(* CoDeSys 2.3.9.41 project: hlor.pro *)
(* Libraries: STANDARD.LIB 4.10.05 11:14:46, IECSFC.LIB 13.4.06 15:51:28, ANALYZATION.LIB 5.10.99 09:05:06 *)

(* PLC configuration (modules and I/O channels)
AT %IX0.0 [BitInput] {ChannellName = Enter name}
AT %IX0.1 [BitInput] {ChannellName = Enter name}
AT %IX0.2 [BitInput] {ChannellName = Enter name}
AT %IX0.3 [BitInput] {ChannellName = Enter name}
AT %IB1.0 [ByteInput] {ChannellName = Enter name}
AT %IB1.1 [ByteInput] {ChannellName = Enter name}
SolNasos AT %QX2.0 [BitOutput] Вкл/Выкл солевого насоса {ChannellName = Enter name}
WaterNasos AT %QX2.1 [BitOutput] Вкл/Выкл насоса воды {ChannellName = Enter name}
Klapan AT %QX2.2 [BitOutput] Вкл/Выкл клапана воды {ChannellName = Enter name}
Elektroliz AT %QX2.3 [BitOutput] Вкл/Выкл выпрямителя {ChannellName = Enter name}
AT %QB3.0 [ByteOutput] {ChannellName = Enter name}
AT %QB3.1 [ByteOutput] {ChannellName = Enter name}
D_Volume_Bak AT %IR4.0 [FloatInputP] Объем бака {ChannellName = Fast analog input; AIN_TYPE = 4-20 mA; Peak_Filtr = 200; Flt_Ch = Off; TauRC = 10; MinFV = 0; MaxFV = 150}
D_Konduktivnost AT %IR4.1 [FloatInputP] D_Konduktivnost {ChannellName = Fast analog input; AIN_TYPE = 4-20 mA; Peak_Filtr = 200; Flt_Ch = Off; TauRC = 10; MinFV = 0; MaxFV = 200}
D_Volt AT %IR4.2 [FloatInputP] Ток выпрямителя {ChannellName = Fast analog input; AIN_TYPE = 4-20 mA; Peak_Filtr = 200; Flt_Ch = Off; TauRC = 10; MinFV = 0; MaxFV = 80}
D_Amper AT %IR4.3 [FloatInputP] Напряжение выпрямителя {ChannellName = Fast analog input; AIN_TYPE = 4-20 mA; Peak_Filtr = 200; Flt_Ch = Off; TauRC = 10; MinFV = 0; MaxFV = 200}
DT_Water_Input AT %IR4.4 [FloatInputP] Температура воды на входе {ChannellName = Fast analog input; AIN_TYPE = 4-20 mA; Peak_Filtr = 200; Flt_Ch = Off; TauRC = 10; MinFV = 0; MaxFV = 100}
DT_Water_output AT %IR4.5 [FloatInputP] Температура воды на выходе {ChannellName = Fast analog input; AIN_TYPE = 4-20 mA; Peak_Filtr = 200; Flt_Ch = Off; TauRC = 10; MinFV = 0; MaxFV = 100}
AT %IR4.6 [FloatInputP] {ChannellName = Fast analog input; AIN_TYPE = 4-20 mA; Peak_Filtr = 200; Flt_Ch = Off; TauRC = 10; MinFV = 0; MaxFV = 100}
AT %IR4.7 [FloatInputP] {ChannellName = Fast analog input; AIN_TYPE = 4-20 mA; Peak_Filtr = 200; Flt_Ch = Off; TauRC = 10; MinFV = 0; MaxFV = 20000.0}
AT %IW4.8 [WordInput] {ChannellName = Enter name}
AT %QR5.0 [FloatOutputP] {ChannellName = Analog output; AOUT_TYPE = 4-20 mA; SafeValueREAL = 0.0}
AT %QR5.1 [FloatOutputP] {ChannellName = Analog output; AOUT_TYPE = 4-20 mA; SafeValueREAL = 0.0}
AT %QR5.2 [FloatOutputP] {ChannellName = Analog output; AOUT_TYPE = 4-20 mA; SafeValueREAL = 0.0}
AT %QR5.3 [FloatOutputP] {ChannellName = Analog output; AOUT_TYPE = 4-20 mA; SafeValueREAL = 0.0}
Special input [ID103] node 6, in %IB6 out %QB6 {ChannellName = Special input}
  AT %IX6.0 [BitInput] {ChannellName = Enter name}
Special output [ID104] node 7, in %IB7 out %QB7 {ChannellName = Special output}
  AT %QX7.0 [BitOutput] {ChannellName = Enter name}
Modbus [MODBUS_ID302] node 0, in %IB8.0 out %QB8.0 {ChannellName = Modbus}
  TCP [TCP_ID221] node 0, in %IB8.0.0 out %QB8.0.0 {ChannellName = TCP; RemotePort = 502; Visibility = No}
8 bits [8Bit] node 1, in %IB8.1 out %QB8.1 {ChannellName = 8 bit}
  AT %QB8.1.0 [ByteOutput] {ChannellName = Enter name}
8 bits [8Bit] node 2, in %IB8.2 out %QB8.2 {ChannellName = 8 bit}
  AT %QB8.2.0 [ByteOutput] {ChannellName = Enter name}
8 bits [8Bit] node 3, in %IB8.3 out %QB8.3 {ChannellName = 8 bit}
  AT %QB8.3.0 [ByteOutput] {ChannellName = Enter name}
8 bits [8Bit] node 4, in %IB8.4 out %QB8.4 {ChannellName = 8 bit}
  AT %QB8.4.0 [ByteOutput] {ChannellName = Enter name}
8 bits [8Bit] node 5, in %IB8.5 out %QB8.5 {ChannellName = 8 bit}
  AT %QB8.5.0 [ByteOutput] {ChannellName = Enter name}
8 bits [8Bit] node 6, in %IB8.6 out %QB8.6 {ChannellName = 8 bit}
  AT %QB8.6.0 [ByteOutput] {ChannellName = Enter name}
Float [Float] node 7, in %IB8.7 out %QB8.7 {ChannellName = float}
  D_Volume_Bak_SPK AT %QD8.7.0 [FloatOutput] {ChannellName = Enter name}
Float [Float] node 8, in %IB8.8 out %QB8.8 {ChannellName = float}
  D_Konduktivnost_SPK AT %QD8.8.0 [FloatOutput] {ChannellName = Enter name}
Float [Float] node 9, in %IB8.9 out %QB8.9 {ChannellName = float}
  D_Volt_SPK AT %QD8.9.0 [FloatOutput] {ChannellName = Enter name}
Float [Float] node 10, in %IB8.10 out %QB8.10 {ChannellName = float}
  D_Amper_SPK AT %QD8.10.0 [FloatOutput] {ChannellName = Enter name}
Float [Float] node 11, in %IB8.11 out %QB8.11 {ChannellName = float}
  DT_Water_Input_SPK AT %QD8.11.0 [FloatOutput] {ChannellName = Enter name}
Float [Float] node 12, in %IB8.12 out %QB8.12 {ChannellName = float}
  DT_Water_output_SPK AT %QD8.12.0 [FloatOutput] {ChannellName = Enter name}
8 bits [8Bit] node 13, in %IB8.13 out %QB8.13 {ChannellName = 8 bit}
  AT %QB8.13.0 [ByteOutput] {ChannellName = Enter name}
8 bits [8Bit] node 14, in %IB8.14 out %QB8.14 {ChannellName = 8 bit}
  AT %QB8.14.0 [ByteOutput] {ChannellName = Enter name}
8 bits [8Bit] node 15, in %IB8.15 out %QB8.15 {ChannellName = 8 bit}
  AT %QB8.15.0 [ByteOutput] {ChannellName = Enter name}
8 bits [8Bit] node 16, in %IB8.16 out %QB8.16 {ChannellName = 8 bit}
  AT %QB8.16.0 [ByteOutput] {ChannellName = Enter name}
*)

(* Task configuration *)
TASK NewTask (PRIORITY := 1, INTERVAL := T#200ms);
	PLC_PRG();
END_TASK

(* Global variable list: Global_Variables *)
VAR_GLOBAL
	PLAY_Elektroliz: BOOL := FALSE;
	StartElectroliz: BOOL := FALSE;
	StopElectroliz: BOOL := FALSE;
	StartKlap: BOOL := FALSE;
	StoptKlap: BOOL := FALSE;
	StartWaterNasos: BOOL := FALSE;
	StopWaterNasos: BOOL := FALSE;
	StartSolNasos: BOOL := FALSE;
	StopSolNasos: BOOL := FALSE;
	StartHlorNasos1: BOOL := FALSE;
	StopHlorNasos1: BOOL := FALSE;
	StartHlorNasos2: BOOL := FALSE;
	StopHlorNasos2: BOOL := FALSE;
	StartVozduh: BOOL := FALSE;
	StopVozduh: BOOL := FALSE;
END_VAR

(* POU PLC_PRG, CFC *)
(*
	Программа управления гипохлоридной установкой
	Контроллер ОВЕН ПЛК-160 M2
	Панель оператора ОВЕН СПК310Р

	В ходе работы программы происходит чтение всех входов/выходов.
	Поочередно запускаются функциональные блоки (файлы слева в меню)
	Основное управление происходит с панели оператора. Каждая переменная привязана к кнопкам в панели и влияет на ход работы установки.
*)


PROGRAM PLC_PRG
VAR

	Electroliz_prg: Electroliz; 				(* Программа управления выпрямителем *)
	Hlorirovanie_prg: Hlorirovanie; 		(* Программа управления первичным и вторичным насосами *)
	SoftWater_prg: SoftWater;			(* Программа управления насосом подачи воды *)
	SolNasos_prg: SolNasos;			(* Программа управления насосом подачи солевого раствора *)
	Vozduh_prg: Vozduh;					(* Программа управления вентилятором-вытяжкой *)
	D_Elektroliz_prg: D_Elektroliz;		(* Программа управления сигналами на вкл/выкл выпрямителя *)

END_VAR
VAR (* helpers for the ST form of the networks *)
	_t97 : WORD;
	_t98 : WORD;
	_t99 : WORD;
	_t100 : WORD;
	_t101 : WORD;
	_t204 : WORD;
END_VAR
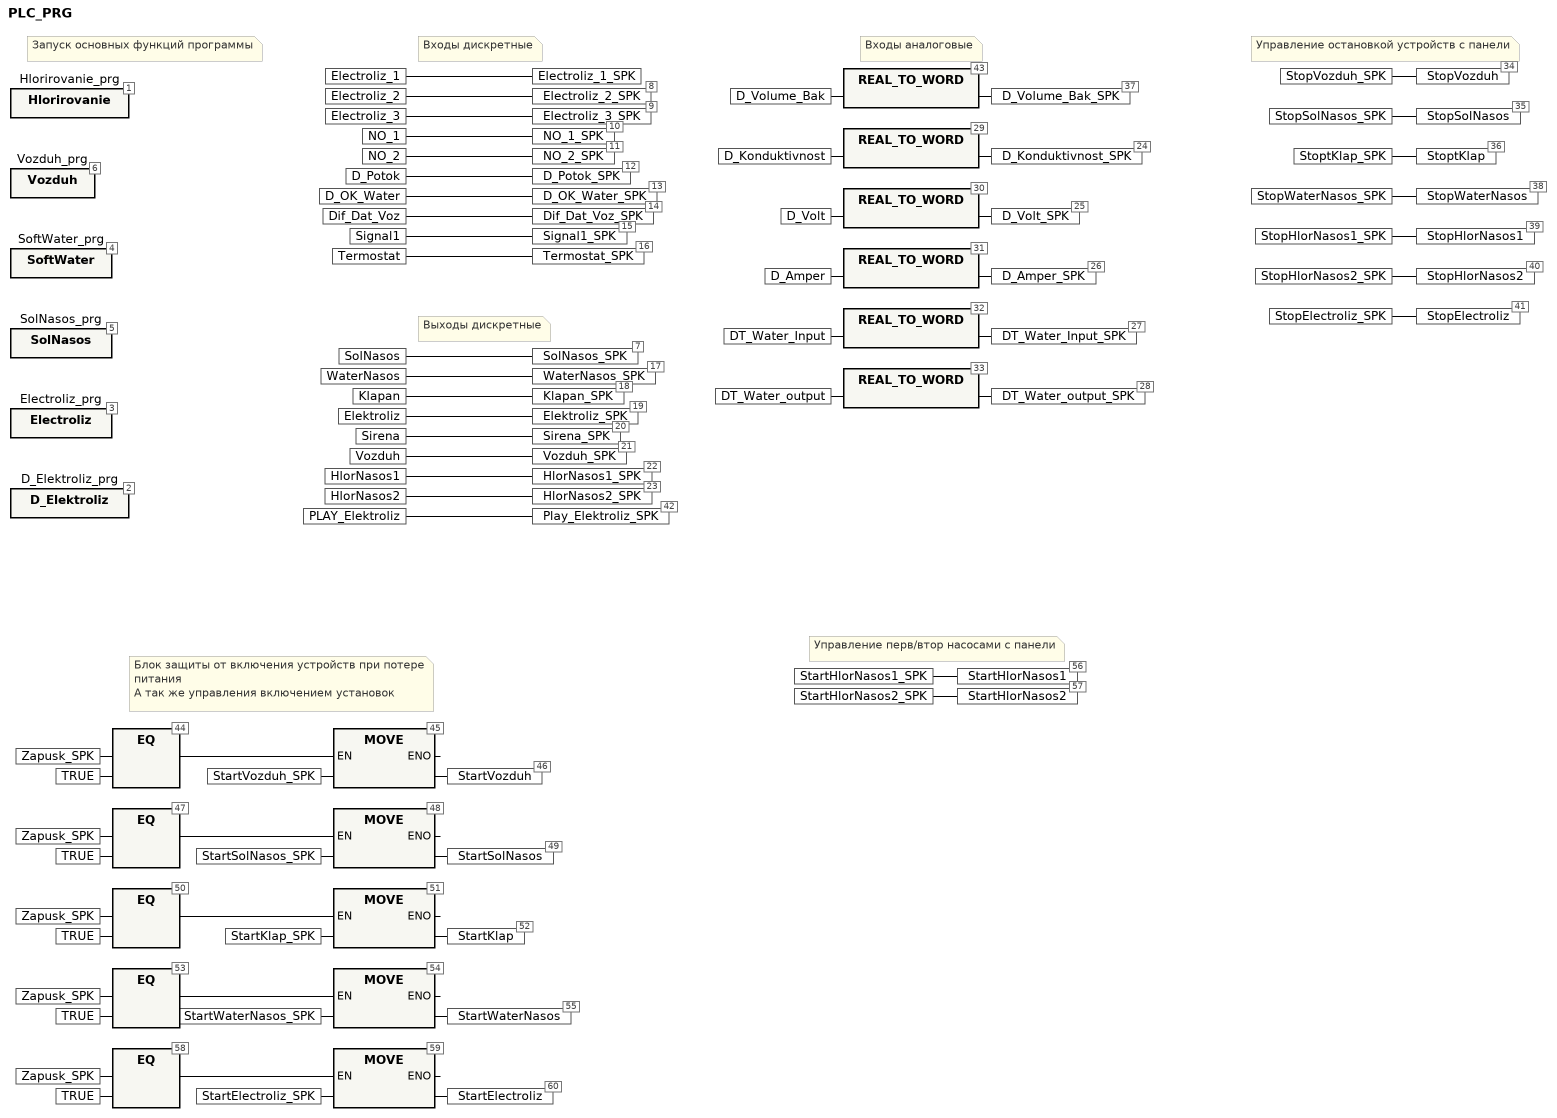
_CFC_ (* Continuous Function Chart, elements in execution order *)
(* Запуск основных функций программы *)
(* Блок защиты от включения устройств при потере питания / А так же управления включением установок *)
#0 Electroliz_1_SPK <= Electroliz_1
#1 Hlorirovanie_prg:Hlorirovanie()
(* Входы дискретные *)
#2 D_Elektroliz_prg:D_Elektroliz()
#3 Electroliz_prg:Electroliz()
#4 SoftWater_prg:SoftWater()
#5 SolNasos_prg:SolNasos()
#6 Vozduh_prg:Vozduh()
(* Выходы дискретные *)
#7 SolNasos_SPK <= SolNasos
#8 Electroliz_2_SPK <= Electroliz_2
#9 Electroliz_3_SPK <= Electroliz_3
#10 NO_1_SPK <= NO_1
#11 NO_2_SPK <= NO_2
#12 D_Potok_SPK <= D_Potok
#13 D_OK_Water_SPK <= D_OK_Water
#14 Dif_Dat_Voz_SPK <= Dif_Dat_Voz
#15 Signal1_SPK <= Signal1
#16 Termostat_SPK <= Termostat
#17 WaterNasos_SPK <= WaterNasos
#18 Klapan_SPK <= Klapan
#19 Elektroliz_SPK <= Elektroliz
#20 Sirena_SPK <= Sirena
#21 Vozduh_SPK <= Vozduh
#22 HlorNasos1_SPK <= HlorNasos1
#23 HlorNasos2_SPK <= HlorNasos2
(* Входы аналоговые *)
#24 D_Konduktivnost_SPK <= #29
#25 D_Volt_SPK <= #30
#26 D_Amper_SPK <= #31
#27 DT_Water_Input_SPK <= #32
#28 DT_Water_output_SPK <= #33
#29 REAL_TO_WORD(D_Konduktivnost)
#30 REAL_TO_WORD(D_Volt)
#31 REAL_TO_WORD(D_Amper)
#32 REAL_TO_WORD(DT_Water_Input)
#33 REAL_TO_WORD(DT_Water_output)
#34 StopVozduh <= StopVozduh_SPK
#35 StopSolNasos <= StopSolNasos_SPK
#36 StoptKlap <= StoptKlap_SPK
#37 D_Volume_Bak_SPK <= #43
#38 StopWaterNasos <= StopWaterNasos_SPK
#39 StopHlorNasos1 <= StopHlorNasos1_SPK
#40 StopHlorNasos2 <= StopHlorNasos2_SPK
#41 StopElectroliz <= StopElectroliz_SPK
#42 Play_Elektroliz_SPK <= PLAY_Elektroliz
#43 REAL_TO_WORD(D_Volume_Bak)
#44 EQ(Zapusk_SPK, TRUE)
#45 MOVE(EN: #44, StartVozduh_SPK)
#46 StartVozduh <= #45
#47 EQ(Zapusk_SPK, TRUE)
#48 MOVE(EN: #47, StartSolNasos_SPK)
#49 StartSolNasos <= #48
#50 EQ(Zapusk_SPK, TRUE)
#51 MOVE(EN: #50, StartKlap_SPK)
#52 StartKlap <= #51
#53 EQ(Zapusk_SPK, TRUE)
#54 MOVE(EN: #53, StartWaterNasos_SPK)
#55 StartWaterNasos <= #54
#56 StartHlorNasos1 <= StartHlorNasos1_SPK
#57 StartHlorNasos2 <= StartHlorNasos2_SPK
#58 EQ(Zapusk_SPK, TRUE)
#59 MOVE(EN: #58, StartElectroliz_SPK)
#60 StartElectroliz <= #59
(* Управление остановкой устройств с панели *)
(* Управление перв/втор насосами с панели *)
_END_CFC_
(* the same logic as Structured Text *)
(* Запуск основных функций программы *)
(* Блок защиты от включения устройств при потере питания / А так же управления включением установок *)
Electroliz_1_SPK := Electroliz_1;
Hlorirovanie_prg();
(* Входы дискретные *)
D_Elektroliz_prg();
Electroliz_prg();
SoftWater_prg();
SolNasos_prg();
Vozduh_prg();
(* Выходы дискретные *)
SolNasos_SPK := SolNasos;
Electroliz_2_SPK := Electroliz_2;
Electroliz_3_SPK := Electroliz_3;
NO_1_SPK := NO_1;
NO_2_SPK := NO_2;
D_Potok_SPK := D_Potok;
D_OK_Water_SPK := D_OK_Water;
Dif_Dat_Voz_SPK := Dif_Dat_Voz;
Signal1_SPK := Signal1;
Termostat_SPK := Termostat;
WaterNasos_SPK := WaterNasos;
Klapan_SPK := Klapan;
Elektroliz_SPK := Elektroliz;
Sirena_SPK := Sirena;
Vozduh_SPK := Vozduh;
HlorNasos1_SPK := HlorNasos1;
HlorNasos2_SPK := HlorNasos2;
(* Входы аналоговые *)
D_Konduktivnost_SPK := _t97;
D_Volt_SPK := _t98;
D_Amper_SPK := _t99;
DT_Water_Input_SPK := _t100;
DT_Water_output_SPK := _t101;
_t97 := REAL_TO_WORD(D_Konduktivnost);
_t98 := REAL_TO_WORD(D_Volt);
_t99 := REAL_TO_WORD(D_Amper);
_t100 := REAL_TO_WORD(DT_Water_Input);
_t101 := REAL_TO_WORD(DT_Water_output);
StopVozduh := StopVozduh_SPK;
StopSolNasos := StopSolNasos_SPK;
StoptKlap := StoptKlap_SPK;
D_Volume_Bak_SPK := _t204;
StopWaterNasos := StopWaterNasos_SPK;
StopHlorNasos1 := StopHlorNasos1_SPK;
StopHlorNasos2 := StopHlorNasos2_SPK;
StopElectroliz := StopElectroliz_SPK;
Play_Elektroliz_SPK := PLAY_Elektroliz;
_t204 := REAL_TO_WORD(D_Volume_Bak);
IF Zapusk_SPK = TRUE THEN StartVozduh := StartVozduh_SPK; END_IF;
IF Zapusk_SPK = TRUE THEN StartSolNasos := StartSolNasos_SPK; END_IF;
IF Zapusk_SPK = TRUE THEN StartKlap := StartKlap_SPK; END_IF;
IF Zapusk_SPK = TRUE THEN StartWaterNasos := StartWaterNasos_SPK; END_IF;
StartHlorNasos1 := StartHlorNasos1_SPK;
StartHlorNasos2 := StartHlorNasos2_SPK;
IF Zapusk_SPK = TRUE THEN StartElectroliz := StartElectroliz_SPK; END_IF;
(* Управление остановкой устройств с панели *)
(* Управление перв/втор насосами с панели *)
END_PROGRAM

(* POU Electroliz, CFC *)
(*
	Управление выпрямителем (электролизером)
	
	Для включения выпрямителя должны быть одновременно включены:
	- вентилятор (Vozduh)
	- солевой насос (SolNasos)
	- открыт клапан подачи воды (Klapan)
	- насос подачи воды (WaterNasos)
	- датчик уровня воды (D_OK_Water) должен давать сигнал по наличию достаточного уровня жидкости
	- датчик потока (D_Potok)  должен давать сигнал на уровне, установленном оператором установки вручную
	- сигнал (PLAY_Elektroliz) должен давать свой сигнал на возможность включения установки. На панели оператора отображается значком FS

	Автоматическое выключение выпрямителя происходит при нажатии оператором кнопки выключения выпрямителя или по одному из сигналов:
	или - отключился вентилятор
	или - отсключился насос подачи солевого раствора
	или - закрылся клапан подачи воды
	или - отключился насос подачи воды
	или - сигнал (PLAY_Elektroliz) дал сигнал на отключение
	или - датчик наличия уровня жидкости  дал сигнал на отключение
	или - датчик потока воды дал сигнал на отключение

	В остальных случаях управление отключением выпрямителя происходит вручную оператором через панель
*)


FUNCTION_BLOCK Electroliz
VAR_INPUT
END_VAR
VAR_OUTPUT
END_VAR
VAR
	SR2: SR; 		(* Триггер на вкл/выкл выпрямителя *)
END_VAR
VAR (* helpers for the ST form of the networks *)
	_t56 : BOOL;
	_t60 : BOOL;
	_t25 : BOOL;
	_t63 : BOOL;
	_t66 : BOOL;
	_t50 : BOOL;
	_t100 : BOOL;
	_t14 : BOOL;
	_t29 : BOOL;
	_t87 : BOOL;
	_t90 : BOOL;
	_t81 : BOOL;
	_t93 : BOOL;
	_t96 : BOOL;
	_t84 : BOOL;
	_t103 : BOOL;
END_VAR
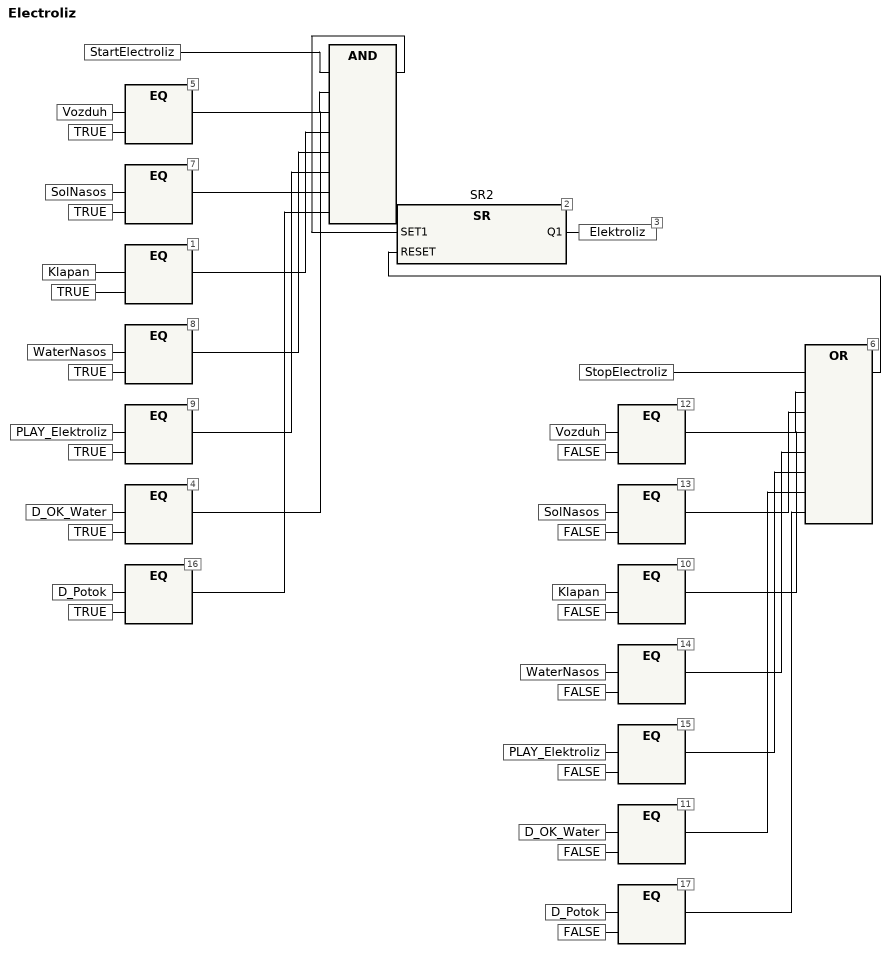
_CFC_ (* Continuous Function Chart, elements in execution order *)
#0 AND(StartElectroliz, #5, #7, #1, #8, #9, #4, #16)
#1 EQ(Klapan, TRUE)
#2 SR2:SR(SET1: #0, RESET: #6)
#3 Elektroliz <= #2.Q1
#4 EQ(D_OK_Water, TRUE)
#5 EQ(Vozduh, TRUE)
#6 OR(StopElectroliz, #12, #13, #10, #14, #15, #11, #17)
#7 EQ(SolNasos, TRUE)
#8 EQ(WaterNasos, TRUE)
#9 EQ(PLAY_Elektroliz, TRUE)
#10 EQ(Klapan, FALSE)
#11 EQ(D_OK_Water, FALSE)
#12 EQ(Vozduh, FALSE)
#13 EQ(SolNasos, FALSE)
#14 EQ(WaterNasos, FALSE)
#15 EQ(PLAY_Elektroliz, FALSE)
#16 EQ(D_Potok, TRUE)
#17 EQ(D_Potok, FALSE)
_END_CFC_
(* the same logic as Structured Text *)
_t14 := StartElectroliz AND _t56 AND _t60 AND _t25 AND _t63 AND _t66 AND _t50 AND _t100;
_t25 := Klapan = TRUE;
SR2(SET1 := _t14, RESET := _t29);
Elektroliz := SR2.Q1;
_t50 := D_OK_Water = TRUE;
_t56 := Vozduh = TRUE;
_t29 := StopElectroliz OR _t87 OR _t90 OR _t81 OR _t93 OR _t96 OR _t84 OR _t103;
_t60 := SolNasos = TRUE;
_t63 := WaterNasos = TRUE;
_t66 := PLAY_Elektroliz = TRUE;
_t81 := Klapan = FALSE;
_t84 := D_OK_Water = FALSE;
_t87 := Vozduh = FALSE;
_t90 := SolNasos = FALSE;
_t93 := WaterNasos = FALSE;
_t96 := PLAY_Elektroliz = FALSE;
_t100 := D_Potok = TRUE;
_t103 := D_Potok = FALSE;
END_FUNCTION_BLOCK

(* POU Vozduh, CFC *)
(*
	Программа включения/выключения вентилятора

	Кнопка StartVoz - при нажатии запускает вентилятор и таймер 5 минут, после истечения времени таймера появляется возможность запуска следующих агрегатов
	Кнопка StopVoz - при нажатии запускает таймер 5 минут, после истечения времени таймера вентилятор выключается. Кнопка выключения заблокирована во время работы других систем

	Включение вентилятора осуществляется в ручном режиме
	Без включенного вентилятора невозможно запустить:
	- насос подачи солевого раствора
	- открыть клапан подачи воды
	- насос подачи воды
	- выпрямитель

	Если вентилятор отключается, то отключаются все остальные устройства
*)


FUNCTION_BLOCK Vozduh
VAR
	SR1: SR; 	(* Триггер на вкл/выкл вентилятора *)
END_VAR
VAR (* helpers for the ST form of the networks *)
	_t106 : BOOL;
	_t124 : BOOL;
	_t120 : BOOL;
END_VAR
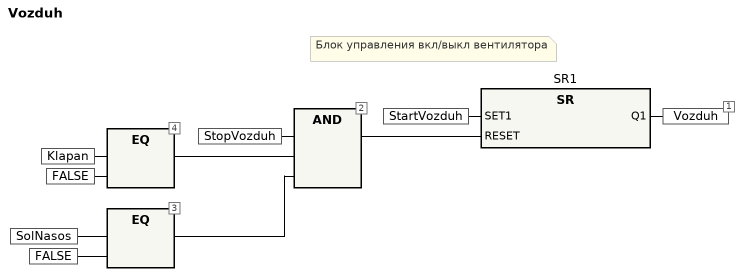
_CFC_ (* Continuous Function Chart, elements in execution order *)
#0 SR1:SR(SET1: StartVozduh, RESET: #2)
#1 Vozduh <= #0.Q1
#2 AND(StopVozduh, #4, #3)
#3 EQ(SolNasos, FALSE)
#4 EQ(Klapan, FALSE)
(* Блок управления вкл/выкл вентилятора *)
_END_CFC_
(* the same logic as Structured Text *)
SR1(SET1 := StartVozduh, RESET := _t106);
Vozduh := SR1.Q1;
_t106 := StopVozduh AND _t124 AND _t120;
_t120 := SolNasos = FALSE;
_t124 := Klapan = FALSE;
(* Блок управления вкл/выкл вентилятора *)
END_FUNCTION_BLOCK

(* POU SolNasos, CFC *)
(*
	Программа включения/выключения солевого насоса

	Кнопка StartSolNasos - производит включение солевого насоса
	Кнопка StopSolNasos - производит выключение солевого насоса

	Для включения насоса солевого раствора должен быть включен вентилятор
	Для отключения необходимо чтобы выпрямитель был отключен
*)


FUNCTION_BLOCK SolNasos
VAR_INPUT
END_VAR
VAR_OUTPUT
END_VAR
VAR
	SR5: SR;	(* Триггер на вкл/выкл насоса подачи солевого раствора *)
END_VAR
VAR (* helpers for the ST form of the networks *)
	_t26 : BOOL;
	_t27 : BOOL;
END_VAR
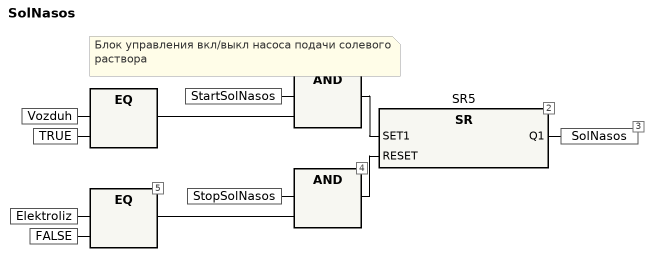
_CFC_ (* Continuous Function Chart, elements in execution order *)
#0 EQ(Vozduh, TRUE)
#1 AND(StartSolNasos, #0)
#2 SR5:SR(SET1: #1, RESET: #4)
#3 SolNasos <= #2.Q1
#4 AND(StopSolNasos, #5)
#5 EQ(Elektroliz, FALSE)
(* Блок управления вкл/выкл насоса подачи солевого раствора *)
_END_CFC_
(* the same logic as Structured Text *)
SR5(SET1 := StartSolNasos AND (Vozduh = TRUE), RESET := _t26);
SolNasos := SR5.Q1;
_t26 := StopSolNasos AND _t27;
_t27 := Elektroliz = FALSE;
(* Блок управления вкл/выкл насоса подачи солевого раствора *)
END_FUNCTION_BLOCK

(* POU Hlorirovanie, CFC *)
(*
	Насосы первичного и вторичного хлорирования
	
	Насосы работют постоянно, независимо от других включенных/выключенных агрегатов
	Выключение насосов производится только в ручном режиме при отключении станции
	Без включенных насосов работа всех остальных агрегатов недопускается
	
	Кнопка StartHlorNasos1 - включает первичный насос хлорирования
	Кнопка StopHlorNasos1 - выключает первичный насос хлорирования
	Кнопка StartHlorNasos2 - включает вторичный насос хлорирования
	Кнопка StopHlorNasos2 - выключает вторичный насос хлорирования
*)


FUNCTION_BLOCK Hlorirovanie
VAR_INPUT
END_VAR
VAR_OUTPUT
END_VAR
VAR
	SR3: SR;	(* Триггер на вкл/выкл первичного насоса хлорирования *)
	SR4: SR;	(* Триггер на вкл/выкл вторичного насоса хлорирования *)
END_VAR
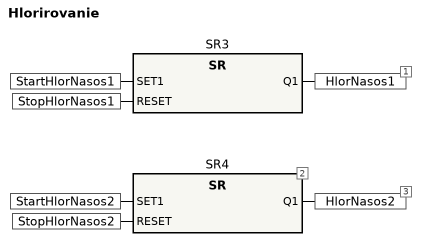
_CFC_ (* Continuous Function Chart, elements in execution order *)
#0 SR3:SR(SET1: StartHlorNasos1, RESET: StopHlorNasos1)
#1 HlorNasos1 <= #0.Q1
#2 SR4:SR(SET1: StartHlorNasos2, RESET: StopHlorNasos2)
#3 HlorNasos2 <= #2.Q1
_END_CFC_
(* the same logic as Structured Text *)
SR3(SET1 := StartHlorNasos1, RESET := StopHlorNasos1);
HlorNasos1 := SR3.Q1;
SR4(SET1 := StartHlorNasos2, RESET := StopHlorNasos2);
HlorNasos2 := SR4.Q1;
END_FUNCTION_BLOCK

(* POU SoftWater, CFC *)
(*
	Управление блоком мягкой воды

	Клапан:
	Кнопка StartKlap -  включение клапана. Кнопка активна только при включенном вентиляторе
	Кнопка StopKlap - выключение клапана. Кнопка активна только при выключенном насосе мягкой воды

	Насос:
	Кнопка StartWaterNasos - включение насоса мягкой воды. Кнопка активна только при включенном клапане
	Кнопка StopWaterNasos	- выключение насоса мягкой воды

	Для включения клапана необходимо наличие включенного вентилятора, без него клапан неоткрывается
	Если клапан открыт, то после можно запускать насос подачи воды
	Если клапан закрыт, то запуск насоса подачи воды невозможен

	Если включен насос подачи воды и включен выпрямитель, то отключение насоса подачи воды, как и клапана, невозможно
	Отключениие устройств при включенном выпрямителе возможно только в случае их технических неисправностей
*)





FUNCTION_BLOCK SoftWater
VAR_INPUT
END_VAR
VAR_OUTPUT
END_VAR
VAR
	SR6: SR;		(* Триггер на вкл/выкл клапана насоса подачи воды *)
	SR7: SR;		(* Триггер на вкл/выкл насоса подачи воды *)
END_VAR
VAR (* helpers for the ST form of the networks *)
	_t25 : BOOL;
	_t24 : BOOL;
	_t32 : BOOL;
	_t40 : BOOL;
	_t43 : BOOL;
	_t47 : BOOL;
	_t48 : BOOL;
END_VAR
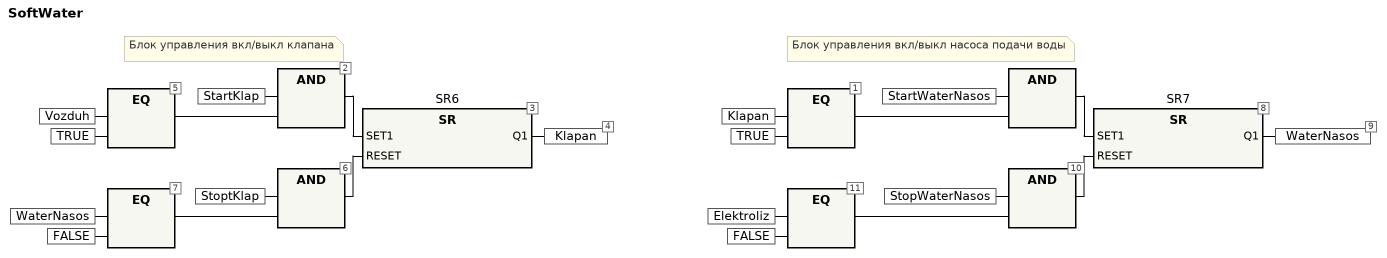
_CFC_ (* Continuous Function Chart, elements in execution order *)
#0 AND(StartWaterNasos, #1)
#1 EQ(Klapan, TRUE)
(* Блок управления вкл/выкл клапана *)
#2 AND(StartKlap, #5)
#3 SR6:SR(SET1: #2, RESET: #6)
#4 Klapan <= #3.Q1
#5 EQ(Vozduh, TRUE)
#6 AND(StoptKlap, #7)
#7 EQ(WaterNasos, FALSE)
#8 SR7:SR(SET1: #0, RESET: #10)
#9 WaterNasos <= #8.Q1
#10 AND(StopWaterNasos, #11)
#11 EQ(Elektroliz, FALSE)
(* Блок управления вкл/выкл насоса подачи воды *)
_END_CFC_
(* the same logic as Structured Text *)
_t24 := StartWaterNasos AND _t25;
_t25 := Klapan = TRUE;
(* Блок управления вкл/выкл клапана *)
SR6(SET1 := StartKlap AND _t32, RESET := _t40);
Klapan := SR6.Q1;
_t32 := Vozduh = TRUE;
_t40 := StoptKlap AND _t43;
_t43 := WaterNasos = FALSE;
SR7(SET1 := _t24, RESET := _t47);
WaterNasos := SR7.Q1;
_t47 := StopWaterNasos AND _t48;
_t48 := Elektroliz = FALSE;
(* Блок управления вкл/выкл насоса подачи воды *)
END_FUNCTION_BLOCK

(* POU D_Elektroliz, CFC *)
(*
	D_Potok - датчик потока воды
	SolNasos - насос подачи солевого раствора
	WaterNasos - насос подачи воды
	PLAY_Elektroliz - сообщается о возможности запуска электролизера, загорается зеленый индикатор LS на дисплее

	Блок включения/выключения выпрямителя (электролизера)
	Включение доступно только при:
	- включенном датчике потока
	- включенном насосе солевого раствора
	- включенном насосе подачи воды
	
	Если датчик потока отключается, то происходит остановка выпрямителя (электролизера).
	Если датчик включен, а затем поток ослабевает, то датчик подает сигнал на выключение выпрямителя
	Если датчик подачи солевого раствора переходит в отключенное состояние, то выпрямитель останавливается
	Если датчик подачи воды показывает, что насос выключен, то выпрямитель останавливается
*)


FUNCTION_BLOCK D_Elektroliz
VAR
	STOP_Elektroliz: BOOL := FALSE;		 (* Переменная выключения выпрямителя в зависимости от состояния датчика потока. По умолчанию в выключенном состоянии *)
END_VAR
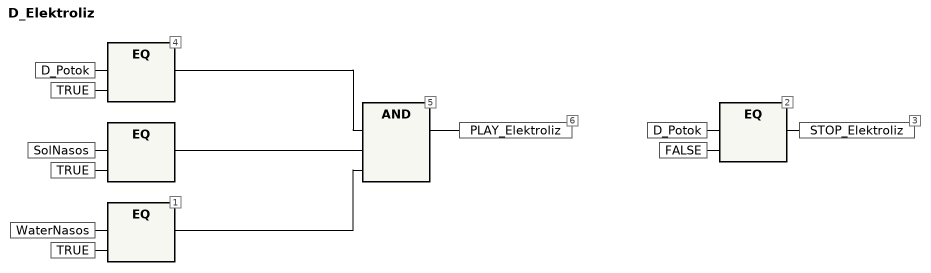
_CFC_ (* Continuous Function Chart, elements in execution order *)
#0 EQ(SolNasos, TRUE)
#1 EQ(WaterNasos, TRUE)
#2 EQ(D_Potok, FALSE)
#3 STOP_Elektroliz <= #2
#4 EQ(D_Potok, TRUE)
#5 AND(#4, #0, #1)
#6 PLAY_Elektroliz <= #5
_END_CFC_
(* the same logic as Structured Text *)
STOP_Elektroliz := D_Potok = FALSE;
PLAY_Elektroliz := (D_Potok = TRUE) AND (SolNasos = TRUE) AND (WaterNasos = TRUE);
END_FUNCTION_BLOCK
